SUBAPPLICATION Uebung_014_AX (* Container (visible/invisible) *)
  (* Standard: 61499-2; Description: Copyright (c) 2023 Meisterschulen am Ostbahnhof This program and the accompanying materials are made available under the terms of the Eclipse Public License 2.0 which is available at https://www.eclipse.org/legal/epl-2.0/ SPDX-License-Identifier: EPL-2.0 *)
  (* Version 1.0, 2023-10-23, Franz Höpfinger, Meisterschulen am Ostbahnhof, initial API and implementation and/or initial documentation *)
  PACKAGE Uebungen;
  IMPORT isobus::UT::io::Softkey::SoftKeyActivationCode::SK_RELEASED;
  IMPORT Uebungen::const::UT::DefaultPool::Container_B;
  IMPORT Uebungen::const::UT::DefaultPool::SoftKey_F1;
  IMPORT Uebungen::const::UT::DefaultPool::SoftKey_F2;
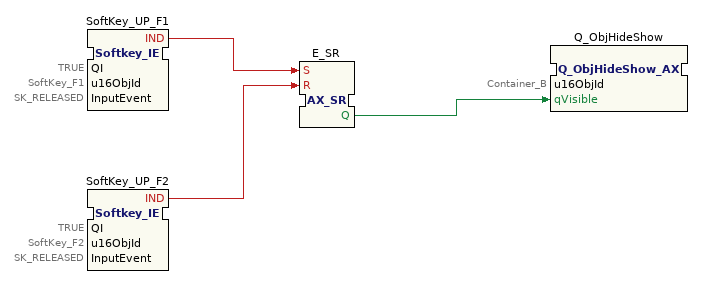
  FBS
    SoftKey_UP_F1 : isobus::UT::io::Softkey::Softkey_IE(QI := TRUE, u16ObjId := SoftKey_F1, InputEvent := SK_RELEASED);
    SoftKey_UP_F2 : isobus::UT::io::Softkey::Softkey_IE(QI := TRUE, u16ObjId := SoftKey_F2, InputEvent := SK_RELEASED);
    E_SR : adapter::events::unidirectional::AX_SR;
    Q_ObjHideShow : isobus::UT::Q::Q_ObjHideShow_AX(u16ObjId := Container_B);
  END_FBS
  EVENT_CONNECTIONS
    SoftKey_UP_F1.IND TO E_SR.S;
    SoftKey_UP_F2.IND TO E_SR.R;
  END_CONNECTIONS
  ADAPTER_CONNECTIONS
    E_SR.Q TO Q_ObjHideShow.qVisible;
  END_CONNECTIONS
END_SUBAPPLICATION
